// TIA Portal V20 export
ORGANIZATION_BLOCK "Cyclic interrupt"   // OB30, FBD, CyclicInterrupt
{ S7_Optimized_Access := 'TRUE' }
// stored: SetENOAutomatically false
   VAR_INPUT
      Initial_Call : Bool;   // Initial call of this OB
      Event_Count : Int;   // Events discarded
   END_VAR
BEGIN

REGION Network 1: Services
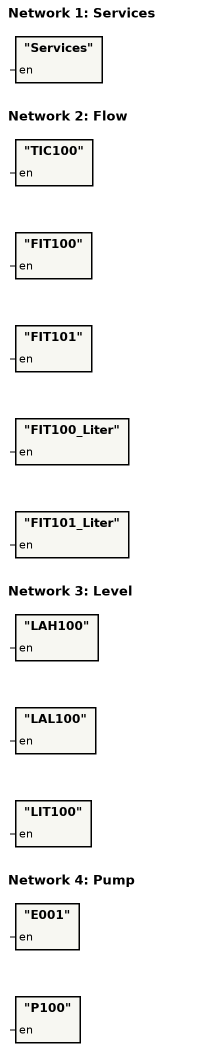
   "Services"();
END_REGION

REGION Network 2: Flow
   "TIC100"();
   "FIT100"();
   "FIT101"();
   "FIT100_Liter"();
   "FIT101_Liter"();
END_REGION

REGION Network 3: Level
   "LAH100"();
   "LAL100"();
   "LIT100"();
END_REGION

REGION Network 4: Pump
   "E001"();
   "P100"();
END_REGION

REGION Network 5: Valve
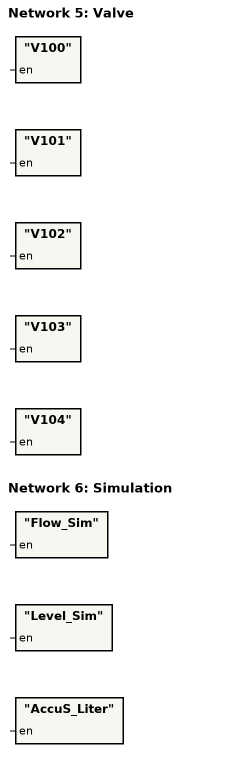
   "V100"();
   "V101"();
   "V102"();
   "V103"();
   "V104"();
END_REGION

REGION Network 6: Simulation
   "Flow_Sim"();
   "Level_Sim"();
   "AccuS_Liter"();
END_REGION
END_ORGANIZATION_BLOCK
